Fanuc KAREL source: kt00341.KL

-- PROVISIONAL review KL for V940-1; original PC SHA256 758aee5a5011f53e371bf9d0922bd8b09fb439956084723dd836b845191c4139
-- Incomplete behavior may be omitted. Consult companion uncertainty JSON. Do not deploy.
PROGRAM KT00341
%NOLOCKGROUP
VAR
  OUT : BOOLEAN
-- UNRESOLVED_DECL Y1 type=002018
-- UNRESOLVED_DECL Y2 type=002018
BEGIN
  -- V9_ZERO_TABLE_METADATA_HINT layout=0001; no indexed target words; source/name/runtime held
  -- UNRESOLVED_PC offsets 5-19; opcodes 2E,22,9D,33,B2
  -- UNRESOLVED_PC offsets 24-38; opcodes 2E,22,9D,33,B2
  -- UNRESOLVED_PC offsets 43-57; opcodes 2E,22,9D,33,B2
  -- UNRESOLVED_PC offsets 62-76; opcodes 2E,22,9D,33,B2
  -- UNRESOLVED_PC offsets 81-106; opcodes 22,9D,33,B1,22,9D,33,B1,59,23
  -- UNRESOLVED_PC offsets 111-115; opcodes 7F
END KT00341
